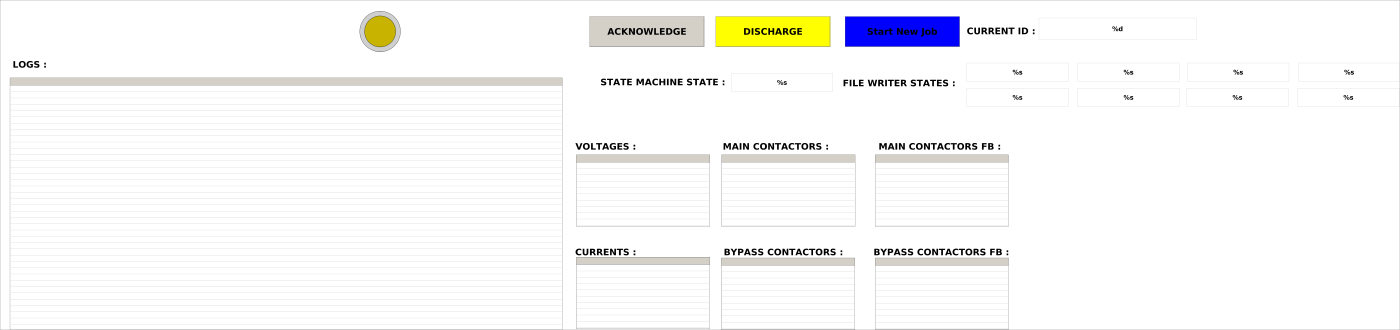
VISUALIZATION Visualisation  // 5552x1312
    Table (39,309 2191x1003), data array: MAIN.sLog
        p3854506369: MAIN.sLog[INDEX]
    Button (2338,65 455x121), "ACKNOWLEDGE", colour toggle: MAIN.b_user_button
        OnMouseDown: execute { MAIN.b_user_button := TRUE; }
        OnMouseUp: execute { MAIN.b_user_button := FALSE; }
    Textfield (2900,291 403x74), "%s", text variable: MAIN.sState
    Label (47,229 340x55), "LOGS :"
    Table (2285,615 530x285), data array: MAIN.n_V_sensors_scaled
        p3854506369: MAIN.n_V_sensors_scaled[INDEX]
    Table (2285,1022 530x285), data array: MAIN.n_A_sensors_scaled
        p3854506369: MAIN.n_A_sensors_scaled[INDEX]
    Label (2279,555 340x55), "VOLTAGES :"
    Label (2278,975 340x55), "CURRENTS :"
    Table (2861,615 530x285), data array: MAIN.b_main_contactors
        p3854506369: MAIN.b_main_contactors[INDEX]
    Label (2863,555 445x55), "MAIN CONTACTORS :"
    Label (2867,975 508x55), "BYPASS CONTACTORS :"
    Table (2860,1025 530x285), data array: MAIN.b_bypass_contactors
        p3854506369: MAIN.b_bypass_contactors[INDEX]
    Table (3470,615 530x285), data array: MAIN.b_main_contactors_fb
        p3854506369: MAIN.b_main_contactors_fb[INDEX]
    Label (3481,555 517x55), "MAIN CONTACTORS FB :"
    Label (3461,975 554x55), "BYPASS CONTACTORS FB :"
    Table (3470,1025 530x285), data array: MAIN.fbMachine.bBypassContactorsFB
        p3854506369: MAIN.fbMachine.bBypassContactorsFB[INDEX]
    Button (2838,65 455x121), "DISCHARGE", colour toggle: MAIN.b_discharge
        OnMouseDown: execute { MAIN.b_discharge :=TRUE; }
        OnMouseUp: execute { MAIN.b_discharge := FALSE; }
    Button (3351,65 455x121), "Start New Job", colour toggle: MAIN.bStartNewJob
        OnMouseDown: execute { MAIN.bStartNewJob := NOT(MAIN.bStartNewJob) }
        OnMouseUp: execute { MAIN.b_discharge := FALSE; }
    Textfield (3834,250 403x74), "%s", text variable: MAIN.s_FBStates[0]
    Textfield (3834,350 403x74), "%s", text variable: MAIN.s_FBStates[2]
    Textfield (4274,250 403x74), "%s", text variable: MAIN.s_FBStates[1]
    Textfield (4274,350 403x74), "%s", text variable: MAIN.s_FBStates[3]
    Label (2378,299 523x55), "STATE MACHINE STATE :"
    Label (3339,303 477x55), "FILE WRITER STATES :"
    Textfield (4120,71 624x87), "%d", text variable: MAIN.nIteration
    Label (3831,96 276x55), "CURRENT ID :"
    Lamp1 (1413,15 189x220), variable: MAIN.b_resetLed, style: Lamp-Lamp1-Yellow
    Textfield (4709,250 403x74), "%s", text variable: MAIN.s_FBStatesContactors[0]
    Textfield (4706,350 403x74), "%s", text variable: MAIN.s_FBStatesContactors[2]
    Textfield (5149,250 403x74), "%s", text variable: MAIN.s_FBStatesContactors[1]
    Textfield (5146,350 403x74), "%s", text variable: MAIN.s_FBStatesContactors[3]
END_VISUALIZATION

(* stored: Version 1.1.0.1, ProductVersion 3.1.4024.12
   Visu Visualisation: Id {13ae7ca4-5b06-4567-966a-d584c9564a1e} *)
